{attribute 'qualified_only'}
//{attribute 'strict'}
{attribute 'to_string'}
TYPE EventsEnum :
(
	NO_EVENT,
	TEST_COMMS, 
	
	//standard operation
	BUNDLE_ETA,
	BUNDLE_IN,
	BUNDLE_OUT,
	BUNDLE_RECEIVED,
	BUNDLE_COMPLETE,
	
	//area complete
	AREA_1_COMPLETE,
	AREA_2_COMPLETE,
	AREA_3_COMPLETE,
	AREA_4_COMPLETE,
	AREA_5_COMPLETE,
	AREA_6_COMPLETE,
	
	//area specific operations
	SECTION_PAPER_COMPLETE,
	SECTION_CARDBOARD_CORNERGUARD_COMPLETE,
	SECTION_CHIPBOARD_COMPLETE,
	SECTION_WOODBUNK_COMPLETE,

	//standard errors
	BACKLOG,
	MACHINE_FAILURE,
	DELAY,
	BUNDLE_EARLY_RECEIVED,
	BUNDLE_LATE_RECEIVED,
	
	//area specific errors
	SECTION_PAPER_FAIL,
	SECTION_CARDBOARD_CORNERGUARD_FAIL,
	SECTION_CHIPBOARD_FAIL,
	SECTION_WOODBUNK_FAIL,
	
	//robots, motors, database, connections, etc
	
	size
);
END_TYPE

(* stored: Version 1.1.0.1, ProductVersion 3.1.4024.11
   EnumerationTextList EventsEnum: Id {7116f09d-954e-4b54-827f-4a9cf285982d} *)
